// TwinCAT 3 PLC project OEF2
// ProgramVersion: 3.1.4024.0
// libraries:
//   Tc2_BABasic, * (Beckhoff Automation GmbH)
//   Tc2_Standard, * (Beckhoff Automation GmbH)
//   Tc2_System, * (Beckhoff Automation GmbH)
//   Tc3_Module, * (Beckhoff Automation GmbH)
// project tree:
//   / GlobalTextList.TcGTLO, PlcTask.TcTTO, Visualization Manager.TcVMO (not stored)
//   POUs/ MAIN.TcPOU
//   VISUs/ Visualization.TcVIS
// real-time tasks:
//   TASK PlcTask: cycle T#10ms, priority 20, ADS port 350
//   TASK PlcTask1: cycle T#10ms, priority 21, ADS port 351

CONFIGURATION OEF2
    RESOURCE PLC ON TwinCAT3
        TASK PlcTask(INTERVAL := T#10ms, PRIORITY := 20);
        PROGRAM MAIN WITH PlcTask : MAIN;
    END_RESOURCE
END_CONFIGURATION

// ---- POUs/MAIN.TcPOU
PROGRAM MAIN
VAR
	iCurrentTemp : INT;
	iSetTemp : INT;
	bheating AT %Q*: BOOL := false;
	iInputsettemp AT %I*: INT;
	iInputcurrenttemp AT %I*: INT;
END_VAR

iSetTemp :=  LREAL_TO_INT(F_Scale(iInputsettemp,0,32767,10,30));
iCurrentTemp :=  LREAL_TO_INT(F_Scale(iInputcurrenttemp,0,32767,-30,40));
IF iSetTemp > iCurrentTemp  THEN
	bheating := TRUE;
ELSE
	bheating := FALSE;
END_IF

END_PROGRAM

// ---- GlobalTextList.TcGTLO
TEXTLIST GlobalTextList
  27 = 'current temp'
  667 = 'current temp %d'
  531 = 'Set temp'
  107 = 'Set temp %D'
  578 = 'Set temp %d'
END_TEXTLIST

// ---- VISUs/Visualization.TcVIS
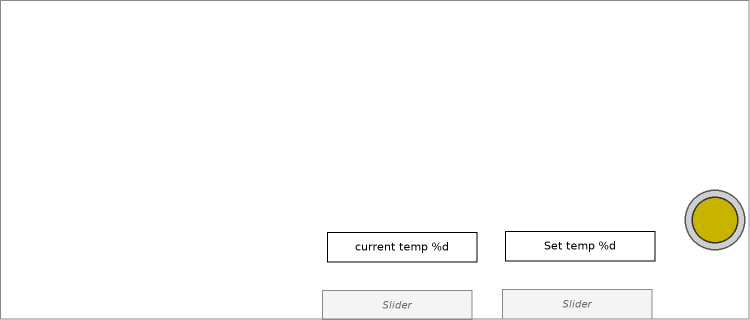
VISUALIZATION Visualization  // 750x320
    Slider (502,289 150x30), variable: MAIN.iInputsettemp, scale 0..32767
    Slider (322,290 150x30), variable: MAIN.iInputcurrenttemp, scale 0..32767
    Lamp1 (680,185 70x70), variable: MAIN.bheating, style: Lamp-Lamp1-Yellow
    Rectangle (327,232 150x30), "current temp %d", text variable: MAIN.iCurrentTemp
    Rectangle (505,231 150x30), "Set temp %d", text variable: MAIN.iSetTemp
END_VISUALIZATION
